FUNCTION_BLOCK Peripherie EXTENDS TcoCore.TcoContext
VAR
	_Handling : Handling(THIS^);
	
END_VAR

(*~
	<docu>
		<summary>
			Main method of the TcoContext. This is the entry point of any control logic that belongs to this context. 
			The call of this method is ensured by calling the <c>InstanceName.Run()</c> method, and it must not be called explicitly.
			This method is abstract, and it must be overridden in derived block.
		</summary>
	</docu>
~*)
METHOD PROTECTED  Main
THIS^.RtcSynchronize(TRUE, '', 60);
_Handling();
END_METHOD

END_FUNCTION_BLOCK

(* stored: Version 1.1.0.1
   POU Peripherie: Id {edd53b5b-305a-41c6-a427-c69c2645d9db}, SpecialFunc None
   Method Main: Id {e000c12e-ec6a-47f9-a04b-64bef24da208} *)
